PROGRAM prgTemperature
VAR
// Kanal 1
	fb_Config_1			: FB_KL320xConfig;
	stInData_1   		AT%I*		: ST_KL320xInData;
	stOutData_1		  	AT%Q*		: ST_KL320xOutData;
// Kanal 2
	fb_Config_2			: FB_KL320xConfig;
	stInData_2   		AT%I*		: ST_KL320xInData;
	stOutData_2  		AT%Q*		: ST_KL320xOutData;

END_VAR

	
	
fb_Config_1(
	bConfigurate:= , 
	bReadConfig:= , 
	iSetSensorType:= , 
	tTimeout:= , 
	bBusy=> , 
	bError=> , 
	iErrorId=> , 
	iState=> , 
	iDataIn=> , 
	iTerminalType=> , 
	iSpecialType=> , 
	iFirmwareVersion=> , 
	sDescription=> , 
	sSensorType=> , 
	bTwoWiredConnection=> , 
	stInData:= stInData_1, 
	stOutData:= stOutData_1);
	
fb_Config_2(
	bConfigurate:= , 
	bReadConfig:= , 
	iSetSensorType:= , 
	tTimeout:= , 
	bBusy=> , 
	bError=> , 
	iErrorId=> , 
	iState=> , 
	iDataIn=> , 
	iTerminalType=> , 
	iSpecialType=> , 
	iFirmwareVersion=> , 
	sDescription=> , 
	sSensorType=> , 
	bTwoWiredConnection=> , 
	stInData:= stInData_2, 
	stOutData:= stOutData_2);

END_PROGRAM

(* stored: Version 1.1.0.1, ProductVersion 3.1.4024.12
   POU prgTemperature: Id {32a15ab6-22ee-4507-9b12-3008b812f0ce}, SpecialFunc None *)
